TYPE
    ST_OutfeedConveyorStatus : STRUCT
        Occupied : USINT;
        Total    : UDINT;
    END_STRUCT
END_TYPE

(* stored: Version 1.1.0.1
   DUT ST_OutfeedConveyorStatus: Id {50bec105-fe1a-414a-b3af-599415a73510} *)
